// TIA Portal V20 export
FUNCTION "ManOperationCm_typeAxis64PosInterface" : Void   // FC80, LAD
// stored: SetENOAutomatically false
   VAR_INPUT
      disableUnit : Bool;
      SoftCamInterface : "LER_typeSoftCamRelation";
   END_VAR
   VAR_OUTPUT
      Status : Word;
      errorID : Word;
   END_VAR
   VAR_IN_OUT
      manualOperationEm : "LAF_typeManEm";
      manualOperationEmArea : "LAF_typeManOperationArea";
      manualOperationCms : "LAF_typeManOperation";
      Axis64Pos : "LBC_typeAxis64PosInterface";
   END_VAR
   VAR_TEMP
      tempMaxPos : LReal;
      tempIndex : Int;
   END_VAR
BEGIN

REGION Network 1 (SCL): MaxPos Find
   FOR #tempIndex := 0 TO 15 DO
       IF #Axis64Pos.configuration.setPositions[#tempIndex].position > #tempMaxPos THEN
           #tempMaxPos := #Axis64Pos.configuration.setPositions[#tempIndex].position;
       END_IF;
   END_FOR;
END_REGION

REGION Network 2: Manual Operation Cm - typeAxis64PosInterface
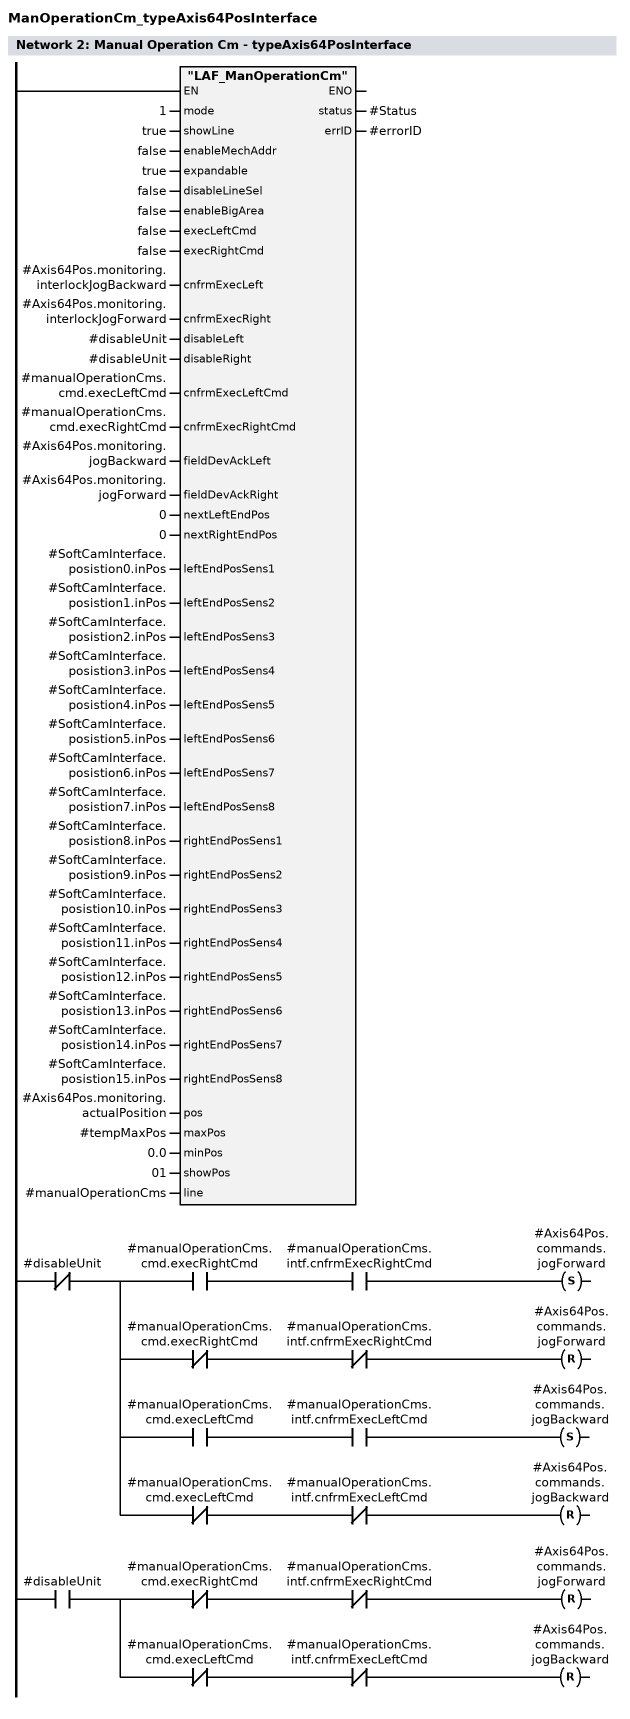
   RUNG wire#powerrail
      "LAF_ManOperationCm"(mode := 1, showLine := true, enableMechAddr := false, expandable := true, disableLineSel := false, enableBigArea := false, execLeftCmd := false, execRightCmd := false, cnfrmExecLeft := #Axis64Pos.monitoring.interlockJogBackward, cnfrmExecRight := #Axis64Pos.monitoring.interlockJogForward, disableLeft := #disableUnit, disableRight := #disableUnit, cnfrmExecLeftCmd := #manualOperationCms.cmd.execLeftCmd, cnfrmExecRightCmd := #manualOperationCms.cmd.execRightCmd, fieldDevAckLeft := #Axis64Pos.monitoring.jogBackward, fieldDevAckRight := #Axis64Pos.monitoring.jogForward, nextLeftEndPos := 0, nextRightEndPos := 0, leftEndPosSens1 := #SoftCamInterface.posistion0.inPos, leftEndPosSens2 := #SoftCamInterface.posistion1.inPos, leftEndPosSens3 := #SoftCamInterface.posistion2.inPos, leftEndPosSens4 := #SoftCamInterface.posistion3.inPos, leftEndPosSens5 := #SoftCamInterface.posistion4.inPos, leftEndPosSens6 := #SoftCamInterface.posistion5.inPos, leftEndPosSens7 := #SoftCamInterface.posistion6.inPos, leftEndPosSens8 := #SoftCamInterface.posistion7.inPos, rightEndPosSens1 := #SoftCamInterface.posistion8.inPos, rightEndPosSens2 := #SoftCamInterface.posistion9.inPos, rightEndPosSens3 := #SoftCamInterface.posistion10.inPos, rightEndPosSens4 := #SoftCamInterface.posistion11.inPos, rightEndPosSens5 := #SoftCamInterface.posistion12.inPos, rightEndPosSens6 := #SoftCamInterface.posistion13.inPos, rightEndPosSens7 := #SoftCamInterface.posistion14.inPos, rightEndPosSens8 := #SoftCamInterface.posistion15.inPos, pos := #Axis64Pos.monitoring.actualPosition, maxPos := #tempMaxPos, minPos := 0.0, showPos := 01, line := #manualOperationCms, status => #Status, errID => #errorID)
   END_RUNG
   RUNG wire#powerrail
      I_Contact( #disableUnit )
      wire#w1
      Contact( #manualOperationCms.cmd.execRightCmd )
      Contact( #manualOperationCms.intf.cnfrmExecRightCmd )
      S_Coil( #Axis64Pos.commands.jogForward )
   END_RUNG
   RUNG wire#w1
      I_Contact( #manualOperationCms.cmd.execRightCmd )
      I_Contact( #manualOperationCms.intf.cnfrmExecRightCmd )
      R_Coil( #Axis64Pos.commands.jogForward )
   END_RUNG
   RUNG wire#w1
      Contact( #manualOperationCms.cmd.execLeftCmd )
      Contact( #manualOperationCms.intf.cnfrmExecLeftCmd )
      S_Coil( #Axis64Pos.commands.jogBackward )
   END_RUNG
   RUNG wire#w1
      I_Contact( #manualOperationCms.cmd.execLeftCmd )
      I_Contact( #manualOperationCms.intf.cnfrmExecLeftCmd )
      R_Coil( #Axis64Pos.commands.jogBackward )
   END_RUNG
   RUNG wire#powerrail
      Contact( #disableUnit )
      wire#w2
      I_Contact( #manualOperationCms.cmd.execRightCmd )
      I_Contact( #manualOperationCms.intf.cnfrmExecRightCmd )
      R_Coil( #Axis64Pos.commands.jogForward )
   END_RUNG
   RUNG wire#w2
      I_Contact( #manualOperationCms.cmd.execLeftCmd )
      I_Contact( #manualOperationCms.intf.cnfrmExecLeftCmd )
      R_Coil( #Axis64Pos.commands.jogBackward )
   END_RUNG
   // the same network as SCL:
   "LAF_ManOperationCm"(mode := 1,
                        showLine := true,
                        enableMechAddr := false,
                        expandable := true,
                        disableLineSel := false,
                        enableBigArea := false,
                        execLeftCmd := false,
                        execRightCmd := false,
                        cnfrmExecLeft := #Axis64Pos.monitoring.interlockJogBackward,
                        cnfrmExecRight := #Axis64Pos.monitoring.interlockJogForward,
                        disableLeft := #disableUnit,
                        disableRight := #disableUnit,
                        cnfrmExecLeftCmd := #manualOperationCms.cmd.execLeftCmd,
                        cnfrmExecRightCmd := #manualOperationCms.cmd.execRightCmd,
                        fieldDevAckLeft := #Axis64Pos.monitoring.jogBackward,
                        fieldDevAckRight := #Axis64Pos.monitoring.jogForward,
                        nextLeftEndPos := 0,
                        nextRightEndPos := 0,
                        leftEndPosSens1 := #SoftCamInterface.posistion0.inPos,
                        leftEndPosSens2 := #SoftCamInterface.posistion1.inPos,
                        leftEndPosSens3 := #SoftCamInterface.posistion2.inPos,
                        leftEndPosSens4 := #SoftCamInterface.posistion3.inPos,
                        leftEndPosSens5 := #SoftCamInterface.posistion4.inPos,
                        leftEndPosSens6 := #SoftCamInterface.posistion5.inPos,
                        leftEndPosSens7 := #SoftCamInterface.posistion6.inPos,
                        leftEndPosSens8 := #SoftCamInterface.posistion7.inPos,
                        rightEndPosSens1 := #SoftCamInterface.posistion8.inPos,
                        rightEndPosSens2 := #SoftCamInterface.posistion9.inPos,
                        rightEndPosSens3 := #SoftCamInterface.posistion10.inPos,
                        rightEndPosSens4 := #SoftCamInterface.posistion11.inPos,
                        rightEndPosSens5 := #SoftCamInterface.posistion12.inPos,
                        rightEndPosSens6 := #SoftCamInterface.posistion13.inPos,
                        rightEndPosSens7 := #SoftCamInterface.posistion14.inPos,
                        rightEndPosSens8 := #SoftCamInterface.posistion15.inPos,
                        pos := #Axis64Pos.monitoring.actualPosition,
                        maxPos := #tempMaxPos,
                        minPos := 0.0,
                        showPos := 01,
                        line := #manualOperationCms,
                        status => #Status,
                        errID => #errorID);
   IF NOT #disableUnit AND #manualOperationCms.cmd.execRightCmd AND #manualOperationCms.intf.cnfrmExecRightCmd THEN
       #Axis64Pos.commands.jogForward := TRUE;
   END_IF;
   IF NOT #disableUnit AND NOT #manualOperationCms.cmd.execRightCmd AND NOT #manualOperationCms.intf.cnfrmExecRightCmd THEN
       #Axis64Pos.commands.jogForward := FALSE;
   END_IF;
   IF NOT #disableUnit AND #manualOperationCms.cmd.execLeftCmd AND #manualOperationCms.intf.cnfrmExecLeftCmd THEN
       #Axis64Pos.commands.jogBackward := TRUE;
   END_IF;
   IF NOT #disableUnit AND NOT #manualOperationCms.cmd.execLeftCmd AND NOT #manualOperationCms.intf.cnfrmExecLeftCmd THEN
       #Axis64Pos.commands.jogBackward := FALSE;
   END_IF;
   IF #disableUnit AND NOT #manualOperationCms.cmd.execRightCmd AND NOT #manualOperationCms.intf.cnfrmExecRightCmd THEN
       #Axis64Pos.commands.jogForward := FALSE;
   END_IF;
   IF #disableUnit AND NOT #manualOperationCms.cmd.execLeftCmd AND NOT #manualOperationCms.intf.cnfrmExecLeftCmd THEN
       #Axis64Pos.commands.jogBackward := FALSE;
   END_IF;
END_REGION
END_FUNCTION
